{attribute 'linkalways'} 
{attribute 'no_explicit_call' := 'This FB is a CLASS and must be accessed using methods or properties'}
{attribute 'enable_dynamic_creation'}
FUNCTION_BLOCK Node_F_VN_FillContainer_ITcVnImage EXTENDS VisionNode
VAR
    ipContainer : _ITcVnContainer;
    ipValue : _ITcVnImage;
    hrPrev : _HRESULT(S_OK);
    hresult : _HRESULT(S_OK);
END_VAR

METHOD PUBLIC  Clone : I_Node
VAR
    pNode : POINTER TO Node_F_VN_FillContainer_ITcVnImage;
END_VAR
pNode := __NEW(Node_F_VN_FillContainer_ITcVnImage);
Clone := pNode^;
END_METHOD

METHOD FB_init : BOOL
VAR_INPUT
    bInitRetains : BOOL; // if TRUE, the retain variables are initialized (warm start / cold start)
    bInCopyCode : BOOL;  // if TRUE, the instance afterwards gets moved into the copy code (online change)
END_VAR
AddInput('ipContainer', ipContainer);
AddInput('ipValue', ipValue);
AddInput('hrPrev', hrPrev);
AddOutput('ipContainer', ipContainer);
AddOutput('hresult',hresult);
END_METHOD

METHOD PROTECTED OnExecute : HRESULT
hresult.Value := F_VN_FillContainer_ITcVnImage(
    ipContainer := ipContainer.Value,
    ipValue := ipValue.Value,
    hrPrev:= hrPrev.Value);
END_METHOD

METHOD PUBLIC PreExecutionCheck
VAR_INPUT
    Check : I_PreExecutionChecks;
END_VAR
Check.IsTrue(ipContainer.IsValid, 'ipContainer must be a valid container');
END_METHOD

END_FUNCTION_BLOCK

(* stored: Version 1.1.0.1, ProductVersion 3.1.4024.13
   POU Node_F_VN_FillContainer_ITcVnImage: Id {25f9bfbb-ba75-477b-9ceb-7f846ac4d9c6}, SpecialFunc None
   Folder Constructor: Id {a93f8ce4-bc80-4921-8ded-abd31f0f9232}
   Method Clone: Id {09d7dd63-d771-47cd-842f-26c0ae4905dc}
   Method FB_init: Id {93295587-9385-45d2-a413-dd273e007ff9}
   Method OnExecute: Id {a94d6e7b-ec11-4373-a0c6-022efc4fb6e7}
   Method PreExecutionCheck: Id {cffae331-f86f-453d-bbdc-ed88b2c574bf} *)
